SUBAPPLICATION logiBUS_IXA_BG (* logiBUS_IXA auf logiBUS_QXA (generisch) *)
  (* Standard: 61499-2; Description: Copyright (c) 2023 Meisterschulen am Ostbahnhof This program and the accompanying materials are made available under the terms of the Eclipse Public License 2.0 which is available at https://www.eclipse.org/legal/epl-2.0/ SPDX-License-Identifier: EPL-2.0 *)
  (* Version 1.1, 2026-09-18, Franz Höpfinger, Meisterschulen am Ostbahnhof, logiBUS_IXA.INITO auf logiBUS_IXA.REQ zurueckverdrahtet (Selfloop) - loest nach der Initialisierung sofort einen Service-Request aus, statt auf die erste echte Wertaenderung am Bus zu warten (Fix fuer 'Waiting for handle'-Status direkt nach Boot). *)
  (* Version 1.0, 2023-10-23, Franz Höpfinger, Meisterschulen am Ostbahnhof, initial API and implementation and/or initial documentation *)
  PACKAGE MyLib::sys;
  IMPORT isobus::UT::Q::const::IDs::ID_NULL;
  IMPORT logiBUS::io::DI::logiBUS_DI;
  IMPORT logiBUS::io::DI::logiBUS_DI_S;
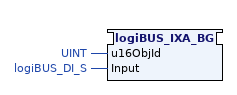
  VAR_INPUT
    u16ObjId : UINT := ID_NULL; (* Object ID *)
    Input : logiBUS::io::DI::logiBUS_DI_S := logiBUS_DI::Invalid; (* Identify the Input Input_I1..I8 *)
  END_VAR
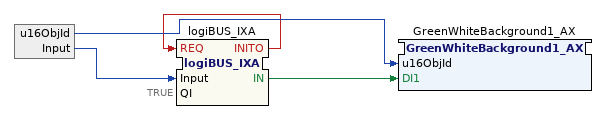
  FBS
    logiBUS_IXA : logiBUS::io::DI::logiBUS_IXA(QI := TRUE);
  END_FBS
  SUBAPPS
    GreenWhiteBackground1_AX : MyLib::sys::GreenWhiteBackground1_AX;
  END_SUBAPPS
  EVENT_CONNECTIONS
    logiBUS_IXA.INITO TO logiBUS_IXA.REQ;
  END_CONNECTIONS
  DATA_CONNECTIONS
    Input TO logiBUS_IXA.Input;
    u16ObjId TO GreenWhiteBackground1_AX.u16ObjId;
  END_CONNECTIONS
  ADAPTER_CONNECTIONS
    logiBUS_IXA.IN TO GreenWhiteBackground1_AX.DI1;
  END_CONNECTIONS
END_SUBAPPLICATION
